Staubli VAL3: onStart.pgx

public program onStart(string& x_sItem[])
begin
  // init all
  bInit=true
end
